Fanuc KAREL source: kt00411.KL

-- PROVISIONAL review KL for V1013-1; original PC SHA256 ab487c30eef611f4164ad1c4eb467595da472535b8edc730fa171535033f150e
-- Incomplete behavior may be omitted. Consult companion uncertainty JSON. Do not deploy.
PROGRAM KT00411
%NOLOCKGROUP
VAR
  I2 : INTEGER
  OUT : BOOLEAN
-- UNRESOLVED_DECL Y1 type=002018
BEGIN
  -- UNRESOLVED_PC offsets 5-19; opcodes 2E,22,9D,33,B2
  -- UNRESOLVED_PC offsets 24-35; opcodes 2E,23
  -- UNRESOLVED_PC offsets 40-62; opcodes 22,9D,33,B1,21,5B,23
  -- UNRESOLVED_PC offsets 67-71; opcodes 7F
END KT00411
